KUKA KRL data list: Maintenance_FromBarrel.dat

&ACCESS RVP
&REL 8
&COMMENT MAINTENANCE LOCATION
DEFDAT Maintenance_FromBarrel
;FOLD HISTORY
;================================
;= Robot Process
;= and Application Control
;================================
;ENDFOLD (HISTORY)
;FOLD EXTERNAL DECLARATIONS
DECL STATE_T STATE,STAT
DECL MODUS_T MODE
DECL INT OFFSET,K,L,M,N,O,KI
;FOLD BAS EXT
EXT  BAS (BAS_COMMAND  :IN,REAL  :IN )
DECL INT SUCCESS
;ENDFOLD (BAS EXT)
;FOLD USER EXT
;Make here your modifictions
;ENDFOLD (USER EXT)
;ENDFOLD (EXTERNAL DECLARATIONS)
DECL FDAT Fhome3={TOOL_NO 1,BASE_NO 0,IPO_FRAME #BASE,POINT2[] " ",TQ_STATE FALSE}
DECL PDAT PPDAT2={VEL 100.000,ACC 5.00000,APO_DIST 100.000,APO_MODE #CDIS,GEAR_JERK 50.0000,EXAX_IGN 0}
DECL BASIS_SUGG_T LAST_BASIS={POINT1[] "P1                      ",POINT2[] "P1                      ",CP_PARAMS[] "CPDAT0                  ",PTP_PARAMS[] "PDAT1                   ",CONT[] "                        ",CP_VEL[] "2.0                     ",PTP_VEL[] "15                      ",SYNC_PARAMS[] "SYNCDAT                 ",SPL_NAME[] "S0                      ",A_PARAMS[] "ADAT0                   "}
DECL E6POS XP1={X 1571.14197,Y -170.537643,Z 294.335754,A -64.2841110,B 86.2638474,C 7.13731289,S 18,T 34,E1 0.0,E2 0.0,E3 0.0,E4 0.0,E5 0.0,E6 0.0}
DECL FDAT FP1={TOOL_NO 1,BASE_NO 0,IPO_FRAME #BASE,POINT2[] " ",TQ_STATE FALSE}
DECL PDAT PPDAT1={VEL 100.000,ACC 100.000,APO_DIST 100.000,APO_MODE #CDIS,GEAR_JERK 50.0000,EXAX_IGN 0}
ENDDAT
